// TIA Portal V16 export
// export: Created 2023-08-28T09:37:43.2617221Z, ExportSetting WithDefaults, DisplayName Totally Integrated Automation Portal, DisplayVersion V16 Update 6, DisplayName TIA Portal Version Control Interface, DisplayVersion V16 Update 2, DisplayName TIA Portal Openness, DisplayVersion V16 Update 6, DisplayName STEP 7 Professional, DisplayVersion V16 Update 6, DisplayName STEP 7 Safety, DisplayVersion V16, DisplayName WinCC Advanced, DisplayVersion V16 Update 6
DATA_BLOCK "SetActivePump_DB_1"   // DB86
AUTHOR : rtecmer
VERSION : 0.1
// stored: AutoNumber true, DBAccessibleFromOPCUA true, InstanceOfName SetActivePump, InstanceOfType FB
"SetActivePump"
   // VAR_IN_OUT
   //    ActivePump : Int;
   //    pumpNum : Int;
   // END_VAR
BEGIN
END_DATA_BLOCK
